// TIA Portal V20 export
ORGANIZATION_BLOCK "Rack or station failure"   // OB86, FBD, RackOrStationFailure
{ S7_Optimized_Access := 'TRUE' }
// stored: SetENOAutomatically false
   VAR_INPUT
      LADDR : HW_DEVICE;   // Hardware identifier
      Event_Class : Byte;   // Event class
      Fault_ID : Byte;   // Fault identifier
   END_VAR
BEGIN

NETWORK
TITLE = call diagnose
      CALL  "Diag", "Diag_DB";

END_ORGANIZATION_BLOCK
